KUKA KRL program: fatgrip.src, fatgrip.dat

--- fatgrip.src ---
&ACCESS RVP
&REL 6
&PARAM EDITMASK = *
&PARAM TEMPLATE = C:\KRC\Roboter\Template\vorgabe
DEF FatGrip( )
;FOLD INI;%{PE}
  ;FOLD BASISTECH INI
    GLOBAL INTERRUPT DECL 3 WHEN $STOPMESS==TRUE DO IR_STOPM ( )
    INTERRUPT ON 3
    BAS (#INITMOV,0 )
  ;ENDFOLD (BASISTECH INI)
;FOLD SPOTTECH INI
USERSPOT(#INIT)
;ENDFOLD (SPOTTECH INI)
;FOLD GRIPPERTECH INI
USER_GRP(0,DUMMY,DUMMY,GDEFAULT)
;ENDFOLD (GRIPPERTECH INI)
  ;FOLD USER INI
    ;Make your modifications here

  ;ENDFOLD (USER INI)
;ENDFOLD (INI)


loop

wait sec 3
closegripper()
wait sec 3

endloop

;FOLD PTP TmrBef Vel=100 % PDAT1 Tool[1]:GripperBP2 Base[0];%{PE}%R 8.3.31,%MKUKATPBASIS,%CMOVE,%VPTP,%P 1:PTP, 2:TmrBef, 3:, 5:100, 7:PDAT1
$BWDSTART=FALSE
PDAT_ACT=PPDAT1
FDAT_ACT=FTmrBef
BAS(#PTP_PARAMS,100)
PTP XTmrBef
;ENDFOLD
;FOLD PTP TmrGrp Vel=100 % PDAT2 Tool[1]:GripperBP2 Base[0];%{PE}%R 8.3.31,%MKUKATPBASIS,%CMOVE,%VPTP,%P 1:PTP, 2:TmrGrp, 3:, 5:100, 7:PDAT2
$BWDSTART=FALSE
PDAT_ACT=PPDAT2
FDAT_ACT=FTmrGrp
BAS(#PTP_PARAMS,100)
PTP XTmrGrp
;ENDFOLD
END

--- fatgrip.dat ---
&ACCESS RVP
&REL 6
&PARAM EDITMASK = *
&PARAM TEMPLATE = C:\KRC\Roboter\Template\vorgabe
DEFDAT  FatGrip
;FOLD EXTERNAL DECLARATIONS;%{PE}%MKUKATPBASIS,%CEXT,%VCOMMON,%P
;FOLD GRIPPERTECH EXT
EXT  H50 (INT  :IN,INT  :IN,INT  :IN,GRP_TYP  :IN )
;ENDFOLD (GRIPPERTECH EXT)
;FOLD SPOTTECH EXT
EXT  USERSPOT (S_COMMAND  :IN,SPOT_TYPE  :IN )
;ENDFOLD (SPOTTECH EXT)
;FOLD BASISTECH EXT;%{PE}%MKUKATPBASIS,%CEXT,%VEXT,%P
EXT  BAS (BAS_COMMAND  :IN,REAL  :IN )
DECL INT SUCCESS
;ENDFOLD (BASISTECH EXT)
;FOLD USER EXT;%{E}%MKUKATPUSER,%CEXT,%VEXT,%P
;Make your modifications here

;ENDFOLD (USER EXT)
;ENDFOLD (EXTERNAL DECLARATIONS)
DECL BASIS_SUGG_T LAST_BASIS={POINT1[] "TmrGrp                  ",POINT2[] "TmrGrp                  ",CP_PARAMS[] "CPDAT0                  ",PTP_PARAMS[] "PDAT2                   ",CONT[] "                        ",CP_VEL[] "2.0                     ",PTP_VEL[] "100                     ",SYNC_PARAMS[] "SYNCDAT                 ",SPL_NAME[] "S0                      ",A_PARAMS[] "ADAT0                   "}
DECL E6POS XTMRBEF={X 1774.48083,Y -2001.86292,Z -617.246887,A 88.1767960,B -2.62970374E-14,C -180.000,S 2,T 42,E1 0.0,E2 0.0,E3 0.0,E4 0.0,E5 0.0,E6 0.0}
DECL FDAT FTmrBef={TOOL_NO 1,BASE_NO 0,IPO_FRAME #BASE,POINT2[] " ",TQ_STATE FALSE}
DECL PDAT PPDAT1={VEL 100.000,ACC 100.000,APO_DIST 100.000,GEAR_JERK 50.0000}
DECL E6POS XTMRGRP={X 1774.48083,Y -2001.86292,Z -1013.76007,A 88.1767960,B -3.84399848E-14,C -180.000,S 2,T 42,E1 0.0,E2 0.0,E3 0.0,E4 0.0,E5 0.0,E6 0.0}
DECL FDAT FTmrGrp={TOOL_NO 1,BASE_NO 0,IPO_FRAME #BASE,POINT2[] " ",TQ_STATE FALSE}
DECL PDAT PPDAT2={VEL 100.000,ACC 100.000,APO_DIST 100.000,GEAR_JERK 50.0000}
ENDDAT
